// TwinCAT 3 PLC project Sortieranlage
// ProgramVersion: 3.1.4026.19
// libraries:
//   Tc2_Standard, * (Beckhoff Automation GmbH)
//   Tc2_System, * (Beckhoff Automation GmbH)
// project tree:
//   DUTs/MachineControl/ E_FactoryOpMode.TcDUT, E_MachineOpMode.TcDUT, E_MachineCommand.TcDUT, ST_MachineControl.TcDUT
//   DUTs/ModuleControl/ E_DirectionSelect.TcDUT
//   DUTs/ModuleStates/ E_ConveyorState.TcDUT, E_ModuleState.TcDUT
//   GVLs/ GVL_Factory.TcGVL
//   / PlcTask.TcTTO
//   POUs/ FB_Conveyor.TcPOU, FB_Distributor.TcPOU, FB_Remover.TcPOU, FB_Feeder.TcPOU, FB_Scale.TcPOU, MAIN.TcPOU
// (motion and I/O tree: see PLC project factoryio)
// real-time tasks:
//   TASK PlcTaskFactoryioConnector: cycle T#5ms, priority 20, ADS port 350
//   TASK PlcTaskSortieranlage: cycle T#10ms, priority 21, ADS port 351
// variable links:
//   (this object) <-> Sortieranlage/Sortieranlage Instance
//     PlcTask Inputs/FactoryioConnector.stOutputs/bAlarmSiren <-> PlcTask Outputs/GVL_Factory.bAlarmSiren
//     PlcTask Inputs/FactoryioConnector.stOutputs/bBtnResetLight <-> PlcTask Outputs/GVL_Factory.bBtnResetLight
//     PlcTask Inputs/FactoryioConnector.stOutputs/bBtnStartLight <-> PlcTask Outputs/GVL_Factory.bBtnStartLight
//     PlcTask Inputs/FactoryioConnector.stOutputs/bBtnStopLight <-> PlcTask Outputs/GVL_Factory.bBtnStopLight
//     PlcTask Inputs/FactoryioConnector.stOutputs/bConveyorFeed <-> PlcTask Outputs/GVL_Factory.bConveyorFeed
//     PlcTask Inputs/FactoryioConnector.stOutputs/bConveyorForward <-> PlcTask Outputs/GVL_Factory.bConveyorForward
//     PlcTask Inputs/FactoryioConnector.stOutputs/bConveyorLeft <-> PlcTask Outputs/GVL_Factory.bConveyorLeft
//     PlcTask Inputs/FactoryioConnector.stOutputs/bConveyorRight <-> PlcTask Outputs/GVL_Factory.bConveyorRight
//     PlcTask Inputs/FactoryioConnector.stOutputs/bConveyorScale <-> PlcTask Outputs/GVL_Factory.bConveyorScale
//     PlcTask Inputs/FactoryioConnector.stOutputs/bEmitter <-> PlcTask Outputs/GVL_Factory.bEmitter
//     PlcTask Inputs/FactoryioConnector.stOutputs/bSorterLeft <-> PlcTask Outputs/GVL_Factory.bSorterLeft
//     PlcTask Inputs/FactoryioConnector.stOutputs/bSorterRaise <-> PlcTask Outputs/GVL_Factory.bSorterRaise
//     PlcTask Inputs/FactoryioConnector.stOutputs/bSorterRight <-> PlcTask Outputs/GVL_Factory.bSorterRight
//     PlcTask Inputs/FactoryioConnector.stOutputs/bStackLightGreen <-> PlcTask Outputs/GVL_Factory.bStackLightGreen
//     PlcTask Inputs/FactoryioConnector.stOutputs/bStackLightRed <-> PlcTask Outputs/GVL_Factory.bStackLightRed
//     PlcTask Inputs/FactoryioConnector.stOutputs/bStackLightYellow <-> PlcTask Outputs/GVL_Factory.bStackLightYellow
//     PlcTask Inputs/FactoryioConnector.stOutputs/nDispCountForward <-> PlcTask Outputs/GVL_Factory.nDispCountForward
//     PlcTask Inputs/FactoryioConnector.stOutputs/nDispCountLeft <-> PlcTask Outputs/GVL_Factory.nDispCountLeft
//     PlcTask Inputs/FactoryioConnector.stOutputs/nDispCountRight <-> PlcTask Outputs/GVL_Factory.nDispCountRight
//     PlcTask Inputs/FactoryioConnector.stOutputs/nDispWeight <-> PlcTask Outputs/GVL_Factory.nDispWeight
//     PlcTask Inputs/FactoryioConnector.stOutputs/nFactoryCameraPosition <-> PlcTask Outputs/GVL_Factory.nFactoryCameraPosition
//     PlcTask Outputs/FactoryioConnector.stInputs/bBtnReset <-> PlcTask Inputs/GVL_Factory.bBtnReset
//     PlcTask Outputs/FactoryioConnector.stInputs/bBtnStart <-> PlcTask Inputs/GVL_Factory.bBtnStart
//     PlcTask Outputs/FactoryioConnector.stInputs/bBtnStopNC <-> PlcTask Inputs/GVL_Factory.bBtnStopNC
//     PlcTask Outputs/FactoryioConnector.stInputs/bFactoryPaused <-> PlcTask Inputs/GVL_Factory.bFactoryPaused
//     PlcTask Outputs/FactoryioConnector.stInputs/bFactoryReset <-> PlcTask Inputs/GVL_Factory.bFactoryReset
//     PlcTask Outputs/FactoryioConnector.stInputs/bFactoryRunning <-> PlcTask Inputs/GVL_Factory.bFactoryRunning
//     PlcTask Outputs/FactoryioConnector.stInputs/bLbConveyorForwardEntry <-> PlcTask Inputs/GVL_Factory.bLbConveyorForwardEntry
//     PlcTask Outputs/FactoryioConnector.stInputs/bLbConveyorForwardExit <-> PlcTask Inputs/GVL_Factory.bLbConveyorForwardExitNC
//     PlcTask Outputs/FactoryioConnector.stInputs/bLbConveyorLeftEntry <-> PlcTask Inputs/GVL_Factory.bLbConveyorLeftEntry
//     PlcTask Outputs/FactoryioConnector.stInputs/bLbConveyorLeftExit <-> PlcTask Inputs/GVL_Factory.bLbConveyorLeftExitNC
//     PlcTask Outputs/FactoryioConnector.stInputs/bLbConveyorRightEntry <-> PlcTask Inputs/GVL_Factory.bLbConveyorRightEntry
//     PlcTask Outputs/FactoryioConnector.stInputs/bLbConveyorRightExit <-> PlcTask Inputs/GVL_Factory.bLbConveyorRightExitNC
//     PlcTask Outputs/FactoryioConnector.stInputs/bLbScale <-> PlcTask Inputs/GVL_Factory.bLbScale
//     PlcTask Outputs/FactoryioConnector.stInputs/bLbScaleEntry <-> PlcTask Inputs/GVL_Factory.bLbScaleEntryNC
//     PlcTask Outputs/FactoryioConnector.stInputs/bLbScaleExit <-> PlcTask Inputs/GVL_Factory.bLbScaleExit
//     PlcTask Outputs/FactoryioConnector.stInputs/bSwAuto <-> PlcTask Inputs/GVL_Factory.bSwAuto
//     PlcTask Outputs/FactoryioConnector.stInputs/bSwConveyorFeedOn <-> PlcTask Inputs/GVL_Factory.bSwConveyorFeedOn
//     PlcTask Outputs/FactoryioConnector.stInputs/bSwConveyorForwardOn <-> PlcTask Inputs/GVL_Factory.bSwConveyorForwardOn
//     PlcTask Outputs/FactoryioConnector.stInputs/bSwConveyorLeftOn <-> PlcTask Inputs/GVL_Factory.bSwConveyorLeftOn
//     PlcTask Outputs/FactoryioConnector.stInputs/bSwConveyorRightOn <-> PlcTask Inputs/GVL_Factory.bSwConveyorRightOn
//     PlcTask Outputs/FactoryioConnector.stInputs/bSwConveyorScaleOn <-> PlcTask Inputs/GVL_Factory.bSwConveyorScaleOn
//     PlcTask Outputs/FactoryioConnector.stInputs/bSwEmergStopNC <-> PlcTask Inputs/GVL_Factory.bSwEmergStopNC
//     PlcTask Outputs/FactoryioConnector.stInputs/bSwManual <-> PlcTask Inputs/GVL_Factory.bSwManual
//     PlcTask Outputs/FactoryioConnector.stInputs/fFactoryTimeScale <-> PlcTask Inputs/GVL_Factory.fFactoryTimeScale
//     PlcTask Outputs/FactoryioConnector.stInputs/fScaleWeight <-> PlcTask Inputs/GVL_Factory.fScaleWeight

CONFIGURATION Sortieranlage
    RESOURCE PLC ON TwinCAT3
        TASK PlcTask(INTERVAL := T#10ms, PRIORITY := 21);
        PROGRAM MAIN WITH PlcTask : MAIN;
    END_RESOURCE
END_CONFIGURATION

// ---- DUTs/MachineControl/E_FactoryOpMode.TcDUT
{attribute 'qualified_only'}
{attribute 'strict'}
{attribute 'to_string'}
TYPE E_FactoryOpMode :
(
    HALTED,
	RUNNING,
    PAUSED,
    RESET
);
END_TYPE

// ---- DUTs/MachineControl/E_MachineOpMode.TcDUT
{attribute 'qualified_only'}
{attribute 'strict'}
{attribute 'to_string'}
TYPE E_MachineOpMode:
(
	AUTOMATIC,
    MANUAL
);
END_TYPE

// ---- DUTs/MachineControl/E_MachineCommand.TcDUT
{attribute 'qualified_only'}
{attribute 'strict'}
{attribute 'to_string'}
TYPE E_MachineCommand :
(
    STOP,
    START
);
END_TYPE

// ---- DUTs/MachineControl/ST_MachineControl.TcDUT
// Machine control
TYPE ST_MachineControl:
STRUCT
    // Machine operating mode
    eMachineOpMode: E_MachineOpMode;
    // Machine command stored
    eMachineCommand: E_MachineCommand;
    // Factory I/O operating mode
    eFactoryOpMode: E_FactoryOpMode;
    // Stop button impulse
    bStop: BOOL;
    // Start button impulse
    bStart: BOOL;
    // Reset button impulse
    bReset: BOOL;
    // Emergency switch
    bEmergStopNC: BOOL;
END_STRUCT
END_TYPE

// ---- DUTs/ModuleControl/E_DirectionSelect.TcDUT
{attribute 'qualified_only'}
{attribute 'strict'}
{attribute 'to_string'}
TYPE E_DirectionSelect:
(
    UNDEFINED := 0,
	FORWARD,
    LEFT,
    RIGHT
);
END_TYPE

// ---- DUTs/ModuleStates/E_ConveyorState.TcDUT
{attribute 'qualified_only'}
{attribute 'strict'}
{attribute 'to_string'}
TYPE E_ConveyorState :
(
	IDLE,
    RUNNING,
    RUNNING_OUT,
    LOCKOUT
);
END_TYPE

// ---- DUTs/ModuleStates/E_ModuleState.TcDUT
{attribute 'qualified_only'}
{attribute 'strict'}
{attribute 'to_string'}
TYPE E_ModuleState :
(
    IDLE,
    SET_DIRECTION,
    MOVE_PART,
    WAIT_FOR_MEASUREMENT,
    EXECUTING_MEASUREMENT,
    WAIT_FOR_FOLLOWER,
    TRANSFER_TO_FOLLOWER,
    CLEAR_CONVEYOR,
    LOCKOUT
);
END_TYPE

// ---- GVLs/GVL_Factory.TcGVL
{attribute 'qualified_only'}
VAR_GLOBAL
    // S0 Reset
    {attribute 'TcLinkTo' := 'TIPC^Factoryio^Factoryio Instance^PlcTask Outputs^FactoryioConnector.stInputs^bBtnReset'}
    bBtnReset AT %I*: BOOL;
    // S1 Start
    {attribute 'TcLinkTo' := 'TIPC^Factoryio^Factoryio Instance^PlcTask Outputs^FactoryioConnector.stInputs^bBtnStart'}
    bBtnStart AT %I*: BOOL;
    // S2 Stop NC
    {attribute 'TcLinkTo' := 'TIPC^Factoryio^Factoryio Instance^PlcTask Outputs^FactoryioConnector.stInputs^bBtnStopNC'}
    bBtnStopNC AT %I*: BOOL;
    // S3 Manual
    {attribute 'TcLinkTo' := 'TIPC^Factoryio^Factoryio Instance^PlcTask Outputs^FactoryioConnector.stInputs^bSwManual'}
    bSwManual AT %I*: BOOL;
    // S4 Auto
    {attribute 'TcLinkTo' := 'TIPC^Factoryio^Factoryio Instance^PlcTask Outputs^FactoryioConnector.stInputs^bSwAuto'}
    bSwAuto AT %I*: BOOL;
    // S5 Emergency stop
    {attribute 'TcLinkTo' := 'TIPC^Factoryio^Factoryio Instance^PlcTask Outputs^FactoryioConnector.stInputs^bSwEmergStopNC'}
    bSwEmergStopNC AT %I*: BOOL;
    // B10 LB: At scale entry
    {attribute 'TcLinkTo' := 'TIPC^Factoryio^Factoryio Instance^PlcTask Outputs^FactoryioConnector.stInputs^bLbScaleEntry'}
    bLbScaleEntryNC AT %I*: BOOL;
    // B11 LB: At scale
    {attribute 'TcLinkTo' := 'TIPC^Factoryio^Factoryio Instance^PlcTask Outputs^FactoryioConnector.stInputs^bLbScale'}
    bLbScale AT %I*: BOOL;
    // B12 LB: At scale exit
    {attribute 'TcLinkTo' := 'TIPC^Factoryio^Factoryio Instance^PlcTask Outputs^FactoryioConnector.stInputs^bLbScaleExit'}
    bLbScaleExit AT %I*: BOOL;
    // B20 LB: At left entry
    {attribute 'TcLinkTo' := 'TIPC^Factoryio^Factoryio Instance^PlcTask Outputs^FactoryioConnector.stInputs^bLbConveyorLeftEntry'}
    bLbConveyorLeftEntry AT %I*: BOOL;
    // B21 LB: At exit left
    {attribute 'TcLinkTo' := 'TIPC^Factoryio^Factoryio Instance^PlcTask Outputs^FactoryioConnector.stInputs^bLbConveyorLeftExit'}
    bLbConveyorLeftExitNC AT %I*: BOOL;
    // B30 LB: At forward entry
    {attribute 'TcLinkTo' := 'TIPC^Factoryio^Factoryio Instance^PlcTask Outputs^FactoryioConnector.stInputs^bLbConveyorForwardEntry'}
    bLbConveyorForwardEntry AT %I*: BOOL;
    // B31 LB: At exit front
    {attribute 'TcLinkTo' := 'TIPC^Factoryio^Factoryio Instance^PlcTask Outputs^FactoryioConnector.stInputs^bLbConveyorForwardExit'}
    bLbConveyorForwardExitNC AT %I*: BOOL;
    // B40 LB: At right entry
    {attribute 'TcLinkTo' := 'TIPC^Factoryio^Factoryio Instance^PlcTask Outputs^FactoryioConnector.stInputs^bLbConveyorRightEntry'}
    bLbConveyorRightEntry AT %I*: BOOL;
    // B41 LB: At exit right
    {attribute 'TcLinkTo' := 'TIPC^Factoryio^Factoryio Instance^PlcTask Outputs^FactoryioConnector.stInputs^bLbConveyorRightExit'}
    bLbConveyorRightExitNC AT %I*: BOOL;
    // S100 Band Einlauf ein
    {attribute 'TcLinkTo' := 'TIPC^Factoryio^Factoryio Instance^PlcTask Outputs^FactoryioConnector.stInputs^bSwConveyorFeedOn'}
    bSwConveyorFeedOn AT %I*: BOOL;
    // S101 Band Auslauf ein
    {attribute 'TcLinkTo' := 'TIPC^Factoryio^Factoryio Instance^PlcTask Outputs^FactoryioConnector.stInputs^bSwConveyorForwardOn'}
    bSwConveyorForwardOn AT %I*: BOOL;
    // S102 Band Auslauf Links ein
    {attribute 'TcLinkTo' := 'TIPC^Factoryio^Factoryio Instance^PlcTask Outputs^FactoryioConnector.stInputs^bSwConveyorLeftOn'}
    bSwConveyorLeftOn AT %I*: BOOL;
    // S103 Band Auslauf Rechts ein
    {attribute 'TcLinkTo' := 'TIPC^Factoryio^Factoryio Instance^PlcTask Outputs^FactoryioConnector.stInputs^bSwConveyorRightOn'}
    bSwConveyorRightOn AT %I*: BOOL;
    // S104 Band Waage ein
    {attribute 'TcLinkTo' := 'TIPC^Factoryio^Factoryio Instance^PlcTask Outputs^FactoryioConnector.stInputs^bSwConveyorScaleOn'}
    bSwConveyorScaleOn AT %I*: BOOL;
    // FACTORY I/O (Running)
    {attribute 'TcLinkTo' := 'TIPC^Factoryio^Factoryio Instance^PlcTask Outputs^FactoryioConnector.stInputs^bFactoryRunning'}
    bFactoryRunning AT %I*: BOOL;
    // FACTORY I/O (Paused)
    {attribute 'TcLinkTo' := 'TIPC^Factoryio^Factoryio Instance^PlcTask Outputs^FactoryioConnector.stInputs^bFactoryPaused'}
    bFactoryPaused AT %I*: BOOL;
    // FACTORY I/O (Reset)
    {attribute 'TcLinkTo' := 'TIPC^Factoryio^Factoryio Instance^PlcTask Outputs^FactoryioConnector.stInputs^bFactoryReset'}
    bFactoryReset AT %I*: BOOL;
    // Gewicht
    {attribute 'TcLinkTo' := 'TIPC^Factoryio^Factoryio Instance^PlcTask Outputs^FactoryioConnector.stInputs^fScaleWeight'}
    fScaleWeight AT %I*: REAL;
    // FACTORY I/O (Time Scale)
    {attribute 'TcLinkTo' := 'TIPC^Factoryio^Factoryio Instance^PlcTask Outputs^FactoryioConnector.stInputs^fFactoryTimeScale'}
    fFactoryTimeScale AT %I*: REAL;

    // H0 Reset light
    {attribute 'TcLinkTo' := 'TIPC^Factoryio^Factoryio Instance^PlcTask Inputs^FactoryioConnector.stOutputs^bBtnResetLight'}
    bBtnResetLight AT %Q*: BOOL;
    // H1 Start light
    {attribute 'TcLinkTo' := 'TIPC^Factoryio^Factoryio Instance^PlcTask Inputs^FactoryioConnector.stOutputs^bBtnStartLight'}
    bBtnStartLight AT %Q*: BOOL;
    // H2 Stop light
    {attribute 'TcLinkTo' := 'TIPC^Factoryio^Factoryio Instance^PlcTask Inputs^FactoryioConnector.stOutputs^bBtnStopLight'}
    bBtnStopLight AT %Q*: BOOL;
    // B0 Alarm Siren
    {attribute 'TcLinkTo' := 'TIPC^Factoryio^Factoryio Instance^PlcTask Inputs^FactoryioConnector.stOutputs^bAlarmSiren'}
    bAlarmSiren AT %Q*: BOOL;
    // H20 Signal Light Red
    {attribute 'TcLinkTo' := 'TIPC^Factoryio^Factoryio Instance^PlcTask Inputs^FactoryioConnector.stOutputs^bStackLightRed'}
    bStackLightRed AT %Q*: BOOL;
    // H21 Signal Light Green
    {attribute 'TcLinkTo' := 'TIPC^Factoryio^Factoryio Instance^PlcTask Inputs^FactoryioConnector.stOutputs^bStackLightGreen'}
    bStackLightGreen AT %Q*: BOOL;
    // H22 Signal Light Yellow
    {attribute 'TcLinkTo' := 'TIPC^Factoryio^Factoryio Instance^PlcTask Inputs^FactoryioConnector.stOutputs^bStackLightYellow'}
    bStackLightYellow AT %Q*: BOOL;
    // M10 Entry conveyor
    {attribute 'TcLinkTo' := 'TIPC^Factoryio^Factoryio Instance^PlcTask Inputs^FactoryioConnector.stOutputs^bConveyorFeed'}
    bConveyorFeed AT %Q*: BOOL;
    // M12 Load scale
    {attribute 'TcLinkTo' := 'TIPC^Factoryio^Factoryio Instance^PlcTask Inputs^FactoryioConnector.stOutputs^bConveyorScale'}
    bConveyorScale AT %Q*: BOOL;
    // M20 Left conveyor
    {attribute 'TcLinkTo' := 'TIPC^Factoryio^Factoryio Instance^PlcTask Inputs^FactoryioConnector.stOutputs^bConveyorLeft'}
    bConveyorLeft AT %Q*: BOOL;
    // M30 Front conveyor
    {attribute 'TcLinkTo' := 'TIPC^Factoryio^Factoryio Instance^PlcTask Inputs^FactoryioConnector.stOutputs^bConveyorForward'}
    bConveyorForward AT %Q*: BOOL;
    // M40 Right conveyor
    {attribute 'TcLinkTo' := 'TIPC^Factoryio^Factoryio Instance^PlcTask Inputs^FactoryioConnector.stOutputs^bConveyorRight'}
    bConveyorRight AT %Q*: BOOL;
    // M50 Send left
    {attribute 'TcLinkTo' := 'TIPC^Factoryio^Factoryio Instance^PlcTask Inputs^FactoryioConnector.stOutputs^bSorterLeft'}
    bSorterLeft AT %Q*: BOOL;
    // M51 Send forward
    {attribute 'TcLinkTo' := 'TIPC^Factoryio^Factoryio Instance^PlcTask Inputs^FactoryioConnector.stOutputs^bSorterRaise'}
    bSorterRaise AT %Q*: BOOL;
    // M52 Send right
    {attribute 'TcLinkTo' := 'TIPC^Factoryio^Factoryio Instance^PlcTask Inputs^FactoryioConnector.stOutputs^bSorterRight'}
    bSorterRight AT %Q*: BOOL;
    // Emitter
    {attribute 'TcLinkTo' := 'TIPC^Factoryio^Factoryio Instance^PlcTask Inputs^FactoryioConnector.stOutputs^bEmitter'}
    bEmitter AT %Q*: BOOL;
    // Gewicht
    {attribute 'TcLinkTo' := 'TIPC^Factoryio^Factoryio Instance^PlcTask Inputs^FactoryioConnector.stOutputs^nDispWeight'}
    nDispWeight AT %Q*: INT;
    // Left count
    {attribute 'TcLinkTo' := 'TIPC^Factoryio^Factoryio Instance^PlcTask Inputs^FactoryioConnector.stOutputs^nDispCountLeft'}
    nDispCountLeft AT %Q*: INT;
    // Forward count
    {attribute 'TcLinkTo' := 'TIPC^Factoryio^Factoryio Instance^PlcTask Inputs^FactoryioConnector.stOutputs^nDispCountForward'}
    nDispCountForward AT %Q*: INT;
    // Right count
    {attribute 'TcLinkTo' := 'TIPC^Factoryio^Factoryio Instance^PlcTask Inputs^FactoryioConnector.stOutputs^nDispCountRight'}
    nDispCountRight AT %Q*: INT;
    // FACTORY I/O (Camera Position)
    {attribute 'TcLinkTo' := 'TIPC^Factoryio^Factoryio Instance^PlcTask Inputs^FactoryioConnector.stOutputs^nFactoryCameraPosition'}
    nFactoryCameraPosition AT %Q*: INT;
END_VAR

// ---- POUs/MAIN.TcPOU
PROGRAM MAIN
VAR
    // Control commands and states
    stMachineControl: ST_MachineControl;

    // Module instance feeder
    fbFeeder: FB_Feeder() := (tMovingTimeout := T#4S);
    // Module instance scale
    fbScale: FB_Scale() := (tRunDownTimeout := T#3S, tMovingTimeout := T#4S, tWeightTimeout := T#2S);
    // Module instance distributor
    {warning disable C0564}
    fbDistributor: FB_Distributor(
        pForward := ADR(aRecipePartsForward),
        nForwardSize := XSIZEOF(aRecipePartsForward),
        pLeft := ADR(aRecipePartsLeft),
        nLeftSize := XSIZEOF(aRecipePartsLeft),
        pRight := ADR(aRecipePartsRight),
        nRightSize := XSIZEOF(aRecipePartsRight)
    ) := (
        tRunDownTimeout := T#1S,
        tMovingTimeout := T#4S,
        eFallbackRemoverDirection := E_DirectionSelect.RIGHT,
        fPartWeightTolerance := 0.1,
        tMovingTimeout := T#5S,
        tRunDownTimeout := T#3S
    );
    {warning restore C0564}
    // Module instance remover conveyor forward
    fbRemoverForward: FB_Remover() := (tRunDownTimeout := T#3S, tMovingTimeout := T#5S);
    // Module instance remover conveyor left
    fbRemoverLeft: FB_Remover() := (tRunDownTimeout := T#3S, tMovingTimeout := T#5S);
    // Module instance remover conveyor right
    fbRemoverRight: FB_Remover() := (tRunDownTimeout := T#3S, tMovingTimeout := T#5S);
END_VAR
VAR PERSISTENT
    // Recipe for required part weight to select forward remover
    aRecipePartsForward: ARRAY[0..6] OF REAL := [1.5, 4.0, 5.0, 7.5];
    // Recipe for required part weight to select left remover
    aRecipePartsLeft: ARRAY[0..6] OF REAL := [3.5];
    // Recipe for required part weight to select right remover
    aRecipePartsRight: ARRAY[0..6] OF REAL := [2.5];

    // Processed parts from forward remover in automatic mode
    nPartCountForward: UINT;
    // Processed parts from left remover in automatic mode
    nPartCountLeft: UINT;
    // Processed parts from right remover in automatic mode
    nPartCountRight: UINT;
END_VAR

MachineControl();

IF stMachineControl.eMachineOpMode = E_MachineOpMode.AUTOMATIC THEN
    Automatic();    
END_IF

MachineStatusDisplay(bForceUpdate := FALSE);

METHOD Automatic
VAR_INPUT
END_VAR
// Enable processing
IF stMachineControl.eMachineCommand = E_MachineCommand.START THEN
    fbFeeder.Enable();
END_IF

// Cyclic calls of function block instances
fbFeeder(
    stMachineControl := stMachineControl,
    bPartAtExit := NOT GVL_Factory.bLbScaleEntryNC,
    bReleasePartTransfer := fbScale.bReadyToReceivePart
);
fbScale(
    stMachineControl := stMachineControl,
    bPartAtEntry := NOT GVL_Factory.bLbScaleEntryNC,
    bPartOnScale := GVL_Factory.bLbScale,
    bPartAtExit := GVL_Factory.bLbScaleExit,
    fWeightIn := GVL_Factory.fScaleWeight,
    bReleasePartTransfer := fbDistributor.bReadyToReceivePart
);
fbDistributor(
	stMachineControl := stMachineControl,
	bPartAtEntry := GVL_Factory.bLbScaleExit,
	bPartAtExitForward := GVL_Factory.bLbConveyorForwardEntry,
	bPartAtExitLeft := GVL_Factory.bLbConveyorLeftEntry,
	bPartAtExitRight := GVL_Factory.bLbConveyorRightEntry,
	bReleasePartTransferForward := fbRemoverForward.bReadyToReceivePart,
	bReleasePartTransferLeft := fbRemoverLeft.bReadyToReceivePart,
	bReleasePartTransferRight := fbRemoverRight.bReadyToReceivePart
);
fbRemoverForward(
    stMachineControl := stMachineControl,
    bPartAtExit := NOT GVL_Factory.bLbConveyorForwardExitNC,
    bPartAtEntry := GVL_Factory.bLbConveyorForwardEntry
);
fbRemoverLeft(
    stMachineControl := stMachineControl,
    bPartAtExit := NOT GVL_Factory.bLbConveyorLeftExitNC,
    bPartAtEntry := GVL_Factory.bLbConveyorLeftEntry
);
fbRemoverRight(
    stMachineControl := stMachineControl,
    bPartAtExit := NOT GVL_Factory.bLbConveyorRightExitNC,
    bPartAtEntry := GVL_Factory.bLbConveyorRightEntry
);

// Call function for part distribution
IF fbScale.bWeightIsUpdated THEN
    fbDistributor.AnnounceNextPart(fWeight := fbScale.fWeightOut);
END_IF

// Increase part processing counter
IF fbRemoverForward.bPartProcessed THEN
    nPartCountForward := nPartCountForward + 1;
END_IF
IF fbRemoverLeft.bPartProcessed THEN
    nPartCountLeft := nPartCountLeft + 1;
END_IF
IF fbRemoverRight.bPartProcessed THEN
    nPartCountRight := nPartCountRight + 1;
END_IF

// Output to actuators
GVL_Factory.bEmitter := fbFeeder.bEmitter;
GVL_Factory.bConveyorFeed := fbFeeder.bConveyorOn;
GVL_Factory.bConveyorScale := fbScale.bConveyorOn;
GVL_Factory.bSorterRaise := fbDistributor.bConveyorOn; 
GVL_Factory.bSorterLeft := fbDistributor.bConveyorToLeft;
GVL_Factory.bSorterRight := fbDistributor.bConveyorToRight; 
GVL_Factory.bConveyorForward := fbRemoverForward.bConveyorOn;
GVL_Factory.bConveyorLeft := fbRemoverLeft.bConveyorOn;
GVL_Factory.bConveyorRight := fbRemoverRight.bConveyorOn;
END_METHOD

METHOD MachineControl
VAR_INPUT
END_VAR
VAR
    // One conveyor is blocked
    bOneConveyorLocked: BOOL;
END_VAR
// Factory operating mode
IF GVL_Factory.bFactoryRunning AND GVL_Factory.bFactoryPaused THEN
    stMachineControl.eFactoryOpMode := E_FactoryOpMode.PAUSED;
ELSIF GVL_Factory.bFactoryRunning THEN
    stMachineControl.eFactoryOpMode := E_FactoryOpMode.RUNNING;
ELSE
    stMachineControl.eFactoryOpMode := E_FactoryOpMode.HALTED;
END_IF

// Factory reset has highest priority
IF GVL_Factory.bFactoryReset THEN
    stMachineControl.eFactoryOpMode := E_FactoryOpMode.RESET;
END_IF

// Machine operating mode
{info 'Currently forced to only automatic mode'}
IF GVL_Factory.bSwAuto OR TRUE THEN
    stMachineControl.eMachineOpMode := E_MachineOpMode.AUTOMATIC;
ELSIF GVL_Factory.bSwManual THEN
    stMachineControl.eMachineOpMode := E_MachineOpMode.MANUAL;
END_IF

// One conveyor is blocked
bOneConveyorLocked := fbFeeder.eConveyorState = E_ConveyorState.LOCKOUT OR
    fbScale.eConveyorState = E_ConveyorState.LOCKOUT OR
    fbDistributor.eConveyorState = E_ConveyorState.LOCKOUT OR
    fbRemoverForward.eConveyorState = E_ConveyorState.LOCKOUT OR
    fbRemoverLeft.eConveyorState = E_ConveyorState.LOCKOUT OR
    fbRemoverRight.eConveyorState = E_ConveyorState.LOCKOUT;

IF bOneConveyorLocked THEN
    GVL_Factory.bStackLightRed := TRUE;

    IF GVL_Factory.bBtnReset THEN
        fbFeeder.Reset();
        fbScale.Reset();
        fbDistributor.Reset();
        fbRemoverForward.Reset();
        fbRemoverLeft.Reset();
        fbRemoverRight.Reset();
    END_IF
ELSE
    GVL_Factory.bStackLightRed := FALSE;
END_IF

// Store last stop/start command
IF NOT GVL_Factory.bBtnStopNC THEN
    stMachineControl.eMachineCommand := E_MachineCommand.STOP;
ELSIF GVL_Factory.bBtnStart THEN
    stMachineControl.eMachineCommand := E_MachineCommand.START;
END_IF

// Hardware buttons to machine control struct
stMachineControl.bStop := NOT GVL_Factory.bBtnStopNC;
stMachineControl.bStart := GVL_Factory.bBtnStart;
stMachineControl.bReset := GVL_Factory.bBtnReset;
stMachineControl.bEmergStopNC := GVL_Factory.bSwEmergStopNC;
END_METHOD

METHOD MachineStatusDisplay
VAR_INPUT
    // Force update of displays
    bForceUpdate: BOOL := FALSE;
END_VAR
// Last part weight in gramms
IF fbScale.bWeightIsUpdated OR bForceUpdate THEN
    GVL_Factory.nDispWeight := REAL_TO_INT(fbScale.fWeightOut * 1000);
END_IF

// Increase part processing counter
IF fbRemoverForward.bPartProcessed OR bForceUpdate THEN
    GVL_Factory.nDispCountForward := UINT_TO_INT(nPartCountForward);
END_IF
IF fbRemoverLeft.bPartProcessed OR bForceUpdate THEN
    GVL_Factory.nDispCountLeft := UINT_TO_INT(nPartCountLeft);
END_IF
IF fbRemoverRight.bPartProcessed OR bForceUpdate THEN
    GVL_Factory.nDispCountRight := UINT_TO_INT(nPartCountRight);
END_IF
END_METHOD

END_PROGRAM

// ---- POUs/FB_Feeder.TcPOU
FUNCTION_BLOCK FB_Feeder EXTENDS FB_Conveyor
VAR_INPUT
    // Follower is ready to receive part
    bReleasePartTransfer: BOOL;
    // Part is at conveyor exit
    bPartAtExit: BOOL;
END_VAR
VAR_OUTPUT
    // Enable part emitter
    bEmitter: BOOL;
END_VAR
VAR
    // Enable processing of parts
    bEnable: BOOL;
    // Current state of feeder
    eStateFeeder: E_ModuleState;
END_VAR

// Cyclic calls of function block instances
SUPER^();

// State machine: feeder
CASE eStateFeeder OF
    E_ModuleState.IDLE:
        SUPER^.Stop(bRunOut := FALSE);
        SUPER^.fbMovingTimeout.IN := FALSE;
        IF bEnable THEN
            bEmitter := TRUE;
            eStateFeeder := E_ModuleState.MOVE_PART;
        ELSE
            bEmitter := FALSE;
        END_IF

    E_ModuleState.MOVE_PART:
        SUPER^.Start();
        SUPER^.fbMovingTimeout.IN := TRUE;
        IF PartAtExit() THEN
            SUPER^.fbMovingTimeout.IN := FALSE;
        END_IF
        IF SUPER^.fbMovingTimeout.Q THEN
            {info 'ToDo: throw error message: Part moving timeout'}
            SUPER^.fbMovingTimeout.IN := FALSE;
            eStateFeeder := E_ModuleState.IDLE;
        END_IF

    E_ModuleState.WAIT_FOR_FOLLOWER:
        SUPER^.Stop(bRunOut := FALSE);
        IF NOT bPartAtExit THEN
            {info 'ToDo: throw message: Part was manual removed'}
            eStateFeeder := E_ModuleState.IDLE;
        END_IF
        IF bReleasePartTransfer THEN
            eStateFeeder := E_ModuleState.TRANSFER_TO_FOLLOWER;
        END_IF

    E_ModuleState.TRANSFER_TO_FOLLOWER:
        SUPER^.Start();
        SUPER^.fbMovingTimeout.IN := TRUE;
        IF NOT bPartAtExit THEN
            SUPER^.fbMovingTimeout.IN := FALSE;
            IF bEnable THEN
                eStateFeeder := E_ModuleState.MOVE_PART;
            ELSE
                eStateFeeder := E_ModuleState.CLEAR_CONVEYOR;
            END_IF
        END_IF
        IF SUPER^.fbMovingTimeout.Q THEN
            {info 'ToDo: throw error message: Part transfer moving timeout'}
            SUPER^.fbMovingTimeout.IN := FALSE;
            eStateFeeder := E_ModuleState.IDLE;
        END_IF

    E_ModuleState.CLEAR_CONVEYOR:
        bEmitter := FALSE;
        SUPER^.fbMovingTimeout.IN := TRUE;
        IF PartAtExit() THEN
            SUPER^.fbMovingTimeout.IN := FALSE;
        END_IF
        IF SUPER^.fbMovingTimeout.Q THEN
            SUPER^.fbMovingTimeout.IN := FALSE;
            eStateFeeder := E_ModuleState.IDLE;
        END_IF
END_CASE

// Unset enable
bEnable := FALSE;

// Current state of feeder
{attribute 'monitoring' := 'variable'}
PROPERTY eModuleState: E_ModuleState
GET
eModuleState := eStateFeeder;
END_GET
END_PROPERTY

// Enable processing of parts
METHOD Enable: BOOL
VAR_INPUT
END_VAR
bEnable := TRUE;
END_METHOD

// Return TRUE if part reach conveyor exit and state machine will go to next step
METHOD PRIVATE PartAtExit: BOOL
VAR_INPUT
END_VAR
IF bPartAtExit AND bReleasePartTransfer THEN
    eStateFeeder := E_ModuleState.TRANSFER_TO_FOLLOWER;
ELSIF bPartAtExit THEN
    eStateFeeder := E_ModuleState.WAIT_FOR_FOLLOWER;
ELSE
    PartAtExit := FALSE;
    RETURN;
END_IF

PartAtExit := TRUE;
END_METHOD

// Part moving timeout
{attribute 'monitoring' := 'call'}
PROPERTY PUBLIC tMovingTimeout : TIME
GET
tMovingTimeout := fbMovingTimeout.PT;
END_GET
SET
fbMovingTimeout.PT := tMovingTimeout;
END_SET
END_PROPERTY

END_FUNCTION_BLOCK

// ---- POUs/FB_Conveyor.TcPOU
FUNCTION_BLOCK ABSTRACT FB_Conveyor
VAR_INPUT
    // Machine control
    stMachineControl: ST_MachineControl;
END_VAR
VAR_OUTPUT
    // Conveyor is not ready and locked
    bError: BOOL;
    // Output to conveyor motor
    bConveyorOn: BOOL;
END_VAR
VAR
    // Part moving timeout
    fbMovingTimeout: TON;
    // Run-down-timeout after normal stop
    fbRunDownTimeout: TOF;
    // Current state of conveyor
    eStateConveyor: E_ConveyorState;
END_VAR

// Cyclic call of timer for moving timeout in derived function block
fbMovingTimeout();

// Cyclic call of timer for run-down-timeout after normal stop
IF fbRunDownTimeout.PT > T#0S THEN
    fbRunDownTimeout();
END_IF

// Emergency stop is active
IF NOT stMachineControl.bEmergStopNC THEN
    eStateConveyor := E_ConveyorState.LOCKOUT;
END_IF


CASE eStateConveyor OF
    E_ConveyorState.IDLE:
        bConveyorOn := FALSE;
        fbRunDownTimeout.IN := FALSE;

    E_ConveyorState.RUNNING:
        bConveyorOn := TRUE;
        fbRunDownTimeout.IN := TRUE;

    E_ConveyorState.RUNNING_OUT:
        fbRunDownTimeout.IN := FALSE;
        IF NOT fbRunDownTimeout.Q OR fbRunDownTimeout.PT = T#0S THEN
            eStateConveyor := E_ConveyorState.IDLE;
        END_IF

    E_ConveyorState.LOCKOUT:
        bConveyorOn := FALSE;
        fbRunDownTimeout.IN := FALSE;
        bError := TRUE;
END_CASE

// Current state of conveyor
{attribute 'monitoring' := 'variable'}
PROPERTY eConveyorState: E_ConveyorState
GET
eConveyorState := eStateConveyor;
END_GET
END_PROPERTY

// Current state of the module
PROPERTY ABSTRACT eModuleState: E_ModuleState
GET
END_GET
END_PROPERTY

METHOD PUBLIC Reset
VAR_INPUT
END_VAR
IF stMachineControl.bEmergStopNC AND eStateConveyor = E_ConveyorState.LOCKOUT THEN
    bError := FALSE;
    eStateConveyor := E_ConveyorState.IDLE;
END_IF
END_METHOD

METHOD PROTECTED Start
VAR_INPUT
END_VAR
IF eStateConveyor = E_ConveyorState.IDLE OR eStateConveyor = E_ConveyorState.RUNNING_OUT THEN
    eStateConveyor := E_ConveyorState.RUNNING;
END_IF
END_METHOD

METHOD PROTECTED Stop
VAR_INPUT
    // Enable timeout before conveyor halt
    bRunOut: BOOL := FALSE;
END_VAR
IF eStateConveyor = E_ConveyorState.RUNNING THEN
    // Stop converyor with timeout before halt
    IF fbRunDownTimeout.PT > T#0S AND bRunOut THEN
        eStateConveyor := E_ConveyorState.RUNNING_OUT;

    // Stop conveyor immediately
    ELSE
        eStateConveyor := E_ConveyorState.IDLE;
    END_IF
END_IF
END_METHOD

// Part moving timeout
{attribute 'monitoring' := 'call'}
PROPERTY PUBLIC tMovingTimeout: TIME
GET
tMovingTimeout := fbMovingTimeout.PT;
END_GET
SET
fbMovingTimeout.PT := tMovingTimeout;
END_SET
END_PROPERTY

// Run-down-timeout after normal stop
{attribute 'monitoring' := 'call'}
PROPERTY PUBLIC tRunDownTimeout: TIME
GET
tRunDownTimeout := fbRunDownTimeout.PT;
END_GET
SET
fbRunDownTimeout.PT := tRunDownTimeout;
END_SET
END_PROPERTY

END_FUNCTION_BLOCK

// ---- POUs/FB_Scale.TcPOU
FUNCTION_BLOCK FB_Scale EXTENDS FB_Conveyor
VAR_INPUT
    // Follower is ready to receive part
    bReleasePartTransfer: BOOL;
    // Part is at conveyor entry
    bPartAtEntry: BOOL;
    // Part is on scale
    bPartOnScale: BOOL;
    // Part is at conveyor exit
    bPartAtExit: BOOL;
    // Current weight at scale
    fWeightIn: REAL;
END_VAR
VAR_OUTPUT
    // Module is ready to receive part
    bReadyToReceivePart: BOOL;
    // Measurement data is refreshed in this cycle
    bWeightIsUpdated: BOOL;
    // Measurement data part weight
    fWeightOut: REAL;
END_VAR
VAR
    // Timeout before store measured weight of part
    fbWeightTimeout: TON;
    // Part is complete on distributor
    fbPartAtDistributor: F_TRIG();
    // Current state of scale
    eStateScale: E_ModuleState;
END_VAR

// Cyclic calls of function block instances
SUPER^();
fbWeightTimeout();
fbPartAtDistributor(CLK := bPartAtExit);

// Default to measurement data has not been updated in this cycle
bWeightIsUpdated := FALSE;

// State machine: 
CASE eStateScale OF
    E_ModuleState.IDLE:
        SUPER^.Stop(bRunOut := TRUE);
        SUPER^.fbMovingTimeout.IN := FALSE;
        bReadyToReceivePart := TRUE;
        fbWeightTimeout.IN := FALSE;
        IF bPartAtEntry THEN
            eStateScale := E_ModuleState.MOVE_PART;
        END_IF

    E_ModuleState.MOVE_PART:
        bReadyToReceivePart := FALSE;
        SUPER^.Start();
        SUPER^.fbMovingTimeout.IN := TRUE;
        IF bPartOnScale THEN
            SUPER^.fbMovingTimeout.IN := FALSE;
            eStateScale := E_ModuleState.WAIT_FOR_MEASUREMENT;
        END_IF
        IF SUPER^.fbMovingTimeout.Q THEN
            {info 'ToDo: throw error message: Part moving timeout'}
            SUPER^.fbMovingTimeout.IN := FALSE;
            eStateScale := E_ModuleState.IDLE;
        END_IF
 
    E_ModuleState.WAIT_FOR_MEASUREMENT:
        SUPER^.Stop(bRunOut := FALSE);
        fbWeightTimeout.IN := TRUE;
        IF fbWeightTimeout.Q THEN
            fbWeightTimeout.IN := FALSE;
            eStateScale := E_ModuleState.EXECUTING_MEASUREMENT;
        END_IF
        IF NOT bPartOnScale THEN
            {info 'ToDo: throw error message: Part has been removed from scale'}
            fbWeightTimeout.IN := FALSE;
            eStateScale := E_ModuleState.IDLE;
        END_IF

    E_ModuleState.EXECUTING_MEASUREMENT:
        IF NOT bPartOnScale THEN
            {info 'ToDo: throw error message: Part has been removed from scale'}
            eStateScale := E_ModuleState.IDLE;
        ELSE
            bWeightIsUpdated := TRUE;
            fWeightOut := fWeightIn;
            IF bReleasePartTransfer THEN
                eStateScale := E_ModuleState.TRANSFER_TO_FOLLOWER;
            ELSE
                eStateScale := E_ModuleState.WAIT_FOR_FOLLOWER;
            END_IF
        END_IF

    E_ModuleState.WAIT_FOR_FOLLOWER:
        IF bReleasePartTransfer THEN
            eStateScale := E_ModuleState.TRANSFER_TO_FOLLOWER;
        END_IF

    E_ModuleState.TRANSFER_TO_FOLLOWER:
        SUPER^.Start();
        SUPER^.fbMovingTimeout.IN := TRUE;
        IF fbPartAtDistributor.Q THEN
            SUPER^.fbMovingTimeout.IN := FALSE;
            eStateScale := E_ModuleState.IDLE;
        END_IF
        IF SUPER^.fbMovingTimeout.Q THEN
            {info 'ToDo: throw error message: Part moving timeout'}
            SUPER^.fbMovingTimeout.IN := FALSE;
            eStateScale := E_ModuleState.IDLE;
        END_IF
END_CASE

// Current state of scale
{attribute 'monitoring' := 'variable'}
PROPERTY eModuleState: E_ModuleState
GET
eModuleState := eStateScale;
END_GET
END_PROPERTY

// Timeout before store measured weight of part
{attribute 'monitoring' := 'call'}
PROPERTY tWeightTimeout : TIME
GET
tWeightTimeout := fbWeightTimeout.PT;
END_GET
SET
fbWeightTimeout.PT := tWeightTimeout;
END_SET
END_PROPERTY

END_FUNCTION_BLOCK

// ---- POUs/FB_Distributor.TcPOU
FUNCTION_BLOCK FB_Distributor EXTENDS FB_Conveyor
VAR_INPUT
    // Part is at conveyor entry
    bPartAtEntry: BOOL;
    // Part is at forward conveyor exit
    bPartAtExitForward: BOOL;
    // Part is at left conveyor exit
    bPartAtExitLeft: BOOL;
    // Part is at right conveyor exit
    bPartAtExitRight: BOOL;
    // Follower left is ready to receive part
    bReleasePartTransferLeft: BOOL;
    // Follower forward is ready to receive part
    bReleasePartTransferForward: BOOL;
    // Follower right is ready to receive part
    bReleasePartTransferRight: BOOL;
END_VAR
VAR_OUTPUT
    // Module is ready to receive part
    bReadyToReceivePart: BOOL;
    // Output to left conveyor
    bConveyorToLeft: BOOL;
    // Output to right conveyor
    bConveyorToRight: BOOL;
END_VAR
VAR
    // Part is fully on remover conveyor
    fbPartAtRemover: F_TRIG();
    // Selected remover direction for next part
    eNextRemoverDirection: E_DirectionSelect;
    // Selected remover direction for current part processed from module
    eCurrentRemoverDirection: E_DirectionSelect;
    // Current state of distributor
    eStateDistributor: E_ModuleState;

    // Pointer to recipe for required part weight to select forward remover
    pPartsForward: POINTER TO REAL;
    // Length of recipe array
    nPartsForwardLength: __UXINT;
    // Pointer to recipe for required part weight to select left remover
    pPartsLeft: POINTER TO REAL;
    // Length of recipe array
    nPartsLeftLength: __UXINT;
    // Pointer to recipe for required part weight to select right remover
    pPartsRight: POINTER TO REAL;
    // Length of recipe array
    nPartsRightLength: __UXINT;

    // Tolerated weight deviation
    {attribute 'hide'}
    _fPartWeightTolerance: REAL;
    // Fallback remover direction if weight is not in recipe
    {attribute 'hide'}
    _eFallbackRemoverDirection: E_DirectionSelect;
END_VAR
VAR_TEMP
    // Follower is ready to receive part
    bReleasePartTransfer: BOOL;
END_VAR

// Based on current direction: determine if part is fully on remover conveyor 
CASE eCurrentRemoverDirection OF
    E_DirectionSelect.FORWARD:
        fbPartAtRemover.CLK := bPartAtExitForward;

    E_DirectionSelect.LEFT:
        fbPartAtRemover.CLK := bPartAtExitLeft;

    E_DirectionSelect.RIGHT:
        fbPartAtRemover.CLK := bPartAtExitRight;
END_CASE

// Cyclic calls of function block instances
SUPER^();
fbPartAtRemover();

// State machine: distributor
CASE eStateDistributor OF
    E_ModuleState.IDLE:
        SUPER^.Stop(bRunOut := TRUE);
        SUPER^.fbMovingTimeout.IN := FALSE;
        bReadyToReceivePart := FALSE;
        IF eNextRemoverDirection <> E_DirectionSelect.UNDEFINED THEN
            eStateDistributor := E_ModuleState.SET_DIRECTION;
        END_IF
        // IF bPartAtEntry THEN
        //     {info 'ToDo: throw warning: unannounced part, moving part to fallback direction'}
        //     eStateDistributor := D_SET_DIRECTION;
        // END_IF

    E_ModuleState.SET_DIRECTION:
        IF eNextRemoverDirection <> E_DirectionSelect.UNDEFINED THEN
            eCurrentRemoverDirection := eNextRemoverDirection;
            eNextRemoverDirection := E_DirectionSelect.UNDEFINED;
        ELSE
            eCurrentRemoverDirection := eFallbackRemoverDirection;
        END_IF

        // Set temporary bReleasePartTransfer based of remover on current remover direction
        CASE eCurrentRemoverDirection OF
            E_DirectionSelect.FORWARD:
                bConveyorToLeft := FALSE;
                bConveyorToRight := FALSE;
                bReleasePartTransfer := bReleasePartTransferForward;

            E_DirectionSelect.LEFT:
                bConveyorToLeft := TRUE;
                bConveyorToRight := FALSE;
                bReleasePartTransfer := bReleasePartTransferLeft;

            E_DirectionSelect.RIGHT:
                bConveyorToLeft := FALSE;
                bConveyorToRight := TRUE;
                bReleasePartTransfer := bReleasePartTransferRight;
        END_CASE

        IF bReleasePartTransfer THEN
            bReadyToReceivePart := TRUE;
            eStateDistributor := E_ModuleState.TRANSFER_TO_FOLLOWER;
        ELSE
            eStateDistributor := E_ModuleState.WAIT_FOR_FOLLOWER;
        END_IF

    E_ModuleState.WAIT_FOR_FOLLOWER:
        // Set temporary bReleasePartTransfer based of remover on current remover direction
        CASE eCurrentRemoverDirection OF
            E_DirectionSelect.FORWARD:
                bReleasePartTransfer := bReleasePartTransferForward;

            E_DirectionSelect.LEFT:
                bReleasePartTransfer := bReleasePartTransferLeft;

            E_DirectionSelect.RIGHT:
                bReleasePartTransfer := bReleasePartTransferRight;
        END_CASE

        IF bReleasePartTransfer THEN
            bReadyToReceivePart := TRUE;
            eStateDistributor := E_ModuleState.TRANSFER_TO_FOLLOWER;
        END_IF

    E_ModuleState.TRANSFER_TO_FOLLOWER:
        bReadyToReceivePart := FALSE;
        SUPER^.Start();
        SUPER^.fbMovingTimeout.IN := TRUE;
        IF fbPartAtRemover.Q THEN
            SUPER^.fbMovingTimeout.IN := FALSE;
            eStateDistributor := E_ModuleState.IDLE;
        END_IF
        IF SUPER^.fbMovingTimeout.Q THEN
            {info 'ToDo: throw error message: Part transfer moving timeout'}
            SUPER^.fbMovingTimeout.IN := FALSE;
            eStateDistributor := E_ModuleState.IDLE;
        END_IF
END_CASE

METHOD AnnounceNextPart
VAR_INPUT
    // Weight of next receiving part
    fWeight: REAL;
END_VAR
VAR
    // Lookup index
	nIndex: __UXINT;
END_VAR
// Check recipe to forward remover
nIndex := 0;
WHILE nIndex <= nPartsForwardLength - 1 DO
    // Lookup fWeight in recipe
    IF fWeight >= pPartsForward[nIndex] - fPartWeightTolerance AND fWeight <= pPartsForward[nIndex] + fPartWeightTolerance THEN
        eNextRemoverDirection := E_DirectionSelect.FORWARD;
        RETURN;
    END_IF

    nIndex := nIndex + 1;
END_WHILE

// Check recipe to left remover
nIndex := 0;
WHILE nIndex <= nPartsLeftLength - 1 DO
    // Lookup fWeight in recipe
    IF fWeight >= pPartsLeft[nIndex] - fPartWeightTolerance AND fWeight <= pPartsLeft[nIndex] + fPartWeightTolerance THEN
        eNextRemoverDirection := E_DirectionSelect.LEFT;
        RETURN;
    END_IF

    nIndex := nIndex + 1;
END_WHILE

// Check recipe to right remover
nIndex := 0;
WHILE nIndex <= nPartsRightLength - 1 DO
    // Lookup fWeight in recipe
    IF fWeight >= pPartsRight[nIndex] - fPartWeightTolerance AND fWeight <= pPartsRight[nIndex] + fPartWeightTolerance THEN
        eNextRemoverDirection := E_DirectionSelect.RIGHT;
        RETURN;
    END_IF

    nIndex := nIndex + 1;
END_WHILE

// Given weight is not in recipe, set fallback direction
eNextRemoverDirection := eFallbackRemoverDirection;
{info 'ToDo: throw info message: Fallback remover selected'}
END_METHOD

// Fallback remover direction if weight is not in recipe
{attribute 'monitoring' := 'call'}
PROPERTY eFallbackRemoverDirection: E_DirectionSelect
GET
eFallbackRemoverDirection := _eFallbackRemoverDirection;
END_GET
SET
IF eFallbackRemoverDirection <> E_DirectionSelect.UNDEFINED THEN
    _eFallbackRemoverDirection := eFallbackRemoverDirection;
ELSE
    _eFallbackRemoverDirection := E_DirectionSelect.FORWARD;
END_IF
END_SET
END_PROPERTY

// Current state of distributor
{attribute 'monitoring' := 'variable'}
PROPERTY eModuleState: E_ModuleState
GET
eModuleState := eStateDistributor;
END_GET
END_PROPERTY

// FB_Init is always available implicitly and it is used primarily for initialization.
// The return value is not evaluated. For a specific influence, you can also declare the
// methods explicitly and provide additional code there with the standard initialization
// code. You can evaluate the return value.
METHOD FB_Init: BOOL
VAR_INPUT
    // TRUE: the retain variables are initialized (reset warm / reset cold)
    bInitRetains: BOOL;
    // TRUE: the instance will be copied to the copy code afterward (online change)
    bInCopyCode: BOOL;

    // Contains the address of the recipe array, use the ADR operator to determine the address
    pForward: POINTER TO REAL;
    // Size of the recipe array, use XSIZE operator to determine the size
    nForwardSize: __UXINT;
    // Contains the address of the recipe array, use the ADR operator to determine the address
    pLeft: POINTER TO REAL;
    // Size of the recipe array, use XSIZE operator to determine the size
    nLeftSize: __UXINT;
    // Contains the address of the recipe array, use the ADR operator to determine the address
    pRight: POINTER TO REAL;
    // Size of the recipe array, use XSIZE operator to determine the size
    nRightSize: __UXINT;
END_VAR
VAR CONSTANT
    // REAL size: 4 bytes
    nTypeSize: __UXINT := 4;
END_VAR
// Assign pointers to internal variables
pPartsForward := pForward;
pPartsLeft := pLeft;
pPartsRight := pRight;

// Get number of elements for each recipe array
nPartsForwardLength := nForwardSize / nTypeSize;
nPartsLeftLength := nLeftSize / nTypeSize;
nPartsRightLength := nRightSize / nTypeSize;
END_METHOD

// Tolerated weight deviation
{attribute 'monitoring' := 'call'}
PROPERTY fPartWeightTolerance: REAL
GET
fPartWeightTolerance := _fPartWeightTolerance;
END_GET
SET
_fPartWeightTolerance := fPartWeightTolerance;
END_SET
END_PROPERTY

// Part moving timeout
{attribute 'monitoring' := 'call'}
PROPERTY PUBLIC tMovingTimeout: TIME
GET
tMovingTimeout := fbMovingTimeout.PT;
END_GET
SET
fbMovingTimeout.PT := tMovingTimeout;
END_SET
END_PROPERTY

END_FUNCTION_BLOCK

// ---- POUs/FB_Remover.TcPOU
FUNCTION_BLOCK FB_Remover EXTENDS FB_Conveyor
VAR_INPUT
    // Part is at conveyor entry
    bPartAtEntry: BOOL;
    // Part is at conveyor exit
    bPartAtExit: BOOL;
END_VAR
VAR_OUTPUT
    // Module is ready to receive part
    bReadyToReceivePart: BOOL;
    // Remover processed one part
    bPartProcessed: BOOL;
END_VAR
VAR
    // Part entering remover conveyor
    fbPartAtEntry: R_TRIG();
    // Count parts entering remover conveyor
    nPartsOnConveyor: INT;
    // Current state of remover conveyor
    eStateRemover: E_ModuleState;
END_VAR

// Cyclic calls of function block instances
SUPER^();
fbPartAtEntry(CLK := bPartAtEntry);

// Count parts entering remover conveyor
IF fbPartAtEntry.Q THEN
    nPartsOnConveyor := nPartsOnConveyor + 1;
END_IF

// Default to no part has been processed
bPartProcessed := FALSE;

// State machine: remover
CASE eStateRemover OF
    E_ModuleState.IDLE:
        SUPER^.Stop(bRunOut := TRUE);
        SUPER^.fbMovingTimeout.IN := FALSE;
        bReadyToReceivePart := TRUE;
        IF nPartsOnConveyor > 0 THEN
            eStateRemover := E_ModuleState.MOVE_PART;
        END_IF

    E_ModuleState.MOVE_PART:
        SUPER^.Start();
        SUPER^.fbMovingTimeout.IN := TRUE;
        IF PartAtExit() THEN
            SUPER^.fbMovingTimeout.IN := FALSE;
        END_IF
        IF SUPER^.fbMovingTimeout.Q THEN
            {info 'ToDo: throw error message: Part moving timeout'}
            SUPER^.fbMovingTimeout.IN := FALSE;
            // Reset counter to 0 is moving timeout occurred
            nPartsOnConveyor := 0;
            eStateRemover := E_ModuleState.IDLE;
        END_IF

    E_ModuleState.TRANSFER_TO_FOLLOWER:
        SUPER^.Start();
        SUPER^.fbMovingTimeout.IN := TRUE;
        IF NOT bPartAtExit THEN
            SUPER^.fbMovingTimeout.IN := FALSE;
            // Decrease counter by one part
            nPartsOnConveyor := nPartsOnConveyor - 1;
            // One part has been processed
            bPartProcessed := TRUE;
            IF nPartsOnConveyor > 0 THEN
                eStateRemover := E_ModuleState.MOVE_PART;
            ELSE
                nPartsOnConveyor := 0;
                eStateRemover := E_ModuleState.IDLE;
            END_IF
        END_IF
        IF SUPER^.fbMovingTimeout.Q THEN
            {info 'ToDo: throw error message: Part transfer moving timeout'}
            SUPER^.fbMovingTimeout.IN := FALSE;
            // Reset counter to 0 is moving timeout occurred
            nPartsOnConveyor := 0;
            eStateRemover := E_ModuleState.IDLE;
        END_IF
END_CASE

// Current state of remover conveyor
{attribute 'monitoring' := 'variable'}
PROPERTY eModuleState: E_ModuleState
GET
eModuleState := eStateRemover;
END_GET
END_PROPERTY

// Return TRUE if part reach conveyor exit and state machine will go to next step
METHOD PRIVATE PartAtExit: BOOL
VAR_INPUT
END_VAR
IF bPartAtExit THEN
    eStateRemover := E_ModuleState.TRANSFER_TO_FOLLOWER;
ELSE
    PartAtExit := FALSE;
    RETURN;
END_IF

PartAtExit := TRUE;
END_METHOD

// Maximum duration for part to reach exit of conveyor
{attribute 'monitoring' := 'call'}
PROPERTY PUBLIC tMovingTimeout : TIME
GET
tMovingTimeout := fbMovingTimeout.PT;
END_GET
SET
fbMovingTimeout.PT := tMovingTimeout;
END_SET
END_PROPERTY

END_FUNCTION_BLOCK
